FUNCTION_BLOCK SBCActor (* Combines the SBActor and SBCalibrator function blocks *)
  (* Standard: 61499-2; Description: Requires the http communication layer. *)
  (* Version 1.0, 2017-08-27, Marc Jakobi, HTW Berlin *)
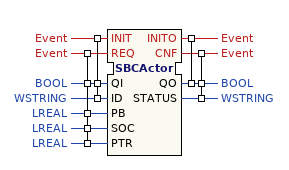
  EVENT_INPUT
    INIT WITH QI, ID; (* Initialization Request *)
    REQ WITH QI, PB, SOC, PTR; (* Normal Execution Request *)
  END_EVENT
  EVENT_OUTPUT
    INITO WITH QO; (* Initialization Confirm *)
    CNF WITH QO, STATUS; (* Execution Confirmation *)
  END_EVENT
  VAR_INPUT
    QI : BOOL; (* Input event qualifier *)
    ID : WSTRING; (* Connection identifier (ip:port) *)
    PB : LREAL; (* Battery transfer (positive = charge, negative = discharge) in W *)
    SOC : LREAL; (* State of charge [0,..,1] *)
    PTR : LREAL; (* Power used to release from trickle charge in W *)
  END_VAR
  VAR_OUTPUT
    QO : BOOL; (* Output event qualifier *)
    STATUS : WSTRING; (* HTTP response codes *)
  END_VAR
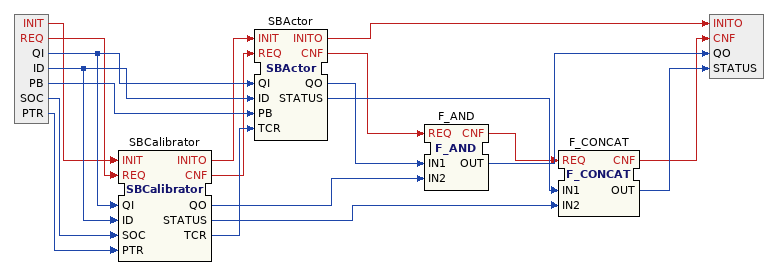
  FBS
    SBActor : SBActor;
    SBCalibrator : SBCalibrator;
    F_AND : F_AND;
    F_CONCAT : F_CONCAT;
  END_FBS
  EVENT_CONNECTIONS
    INIT TO SBCalibrator.INIT;
    SBCalibrator.INITO TO SBActor.INIT;
    SBCalibrator.CNF TO SBActor.REQ;
    SBActor.CNF TO F_AND.REQ;
    SBActor.INITO TO INITO;
    F_AND.CNF TO F_CONCAT.REQ;
    F_CONCAT.CNF TO CNF;
    REQ TO SBCalibrator.REQ;
  END_CONNECTIONS
  DATA_CONNECTIONS
    QI TO SBActor.QI;
    ID TO SBActor.ID;
    ID TO SBCalibrator.ID;
    SBCalibrator.TCR TO SBActor.TCR;
    QI TO SBCalibrator.QI;
    PB TO SBActor.PB;
    SBActor.QO TO F_AND.IN1;
    SBCalibrator.QO TO F_AND.IN2;
    F_AND.OUT TO QO;
    SBActor.STATUS TO F_CONCAT.IN1;
    SBCalibrator.STATUS TO F_CONCAT.IN2;
    F_CONCAT.OUT TO STATUS;
    SOC TO SBCalibrator.SOC;
    PTR TO SBCalibrator.PTR;
  END_CONNECTIONS
END_FUNCTION_BLOCK
